// TIA Portal V16 export
// export: Created 2024-09-05T17:36:33.5266565Z, ExportSetting WithDefaults, DisplayName Totally Integrated Automation Portal, DisplayVersion V16 Update 6, DisplayName TIA Portal Version Control Interface, DisplayVersion V16 Update 2, DisplayName TIA Portal Openness, DisplayVersion V16 Update 6, DisplayName STEP 7 Professional, DisplayVersion V16 Update 6, DisplayName STEP 7 Safety, DisplayVersion V16, DisplayName WinCC Advanced, DisplayVersion V16 Update 6
VAR_GLOBAL   // PLC tag table "hmi"
   iBtnBasicPosition AT %I125.3 : Bool;
   qBasicPosition AT %Q125.1 : Bool;
   qResetAlarm AT %Q125.2 : Bool;
   iBtnResetAlarm AT %I125.4 : Bool;
   iBtnStart AT %I125.2 : Bool;
   qStart AT %Q125.0 : Bool;
   iBtnStartAuto AT %I125.7 : Bool;
   qAuto AT %Q125.3 : Bool;
   qManual AT %Q125.4 : Bool;
   iManual AT %I125.5 : Bool;
   iAuto AT %I125.6 : Bool;
END_VAR
